(* Logix 5000 project; controller RSL5k_18_Template_noLib Emulate 5570 rev 32.11; software revision 32.02; part 16 of 16 *)
(* tags used below, declared in another part *)
   L_TaskMonitor : L_TaskMon[8];

PROGRAM Task_H_MainProgram   (* main routine MainRoutine *)

ROUTINE MainRoutine   (* ladder *)
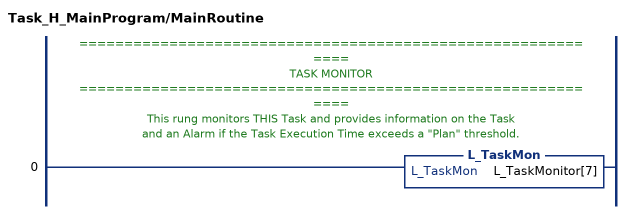
   // ============================================================
   // TASK MONITOR
   // ============================================================
   // This rung monitors THIS Task and provides information on the Task
   // and an Alarm if the Task Execution Time exceeds a "Plan" threshold.
   0: L_TaskMon(L_TaskMonitor[7]);
END_ROUTINE
END_PROGRAM
